// TIA Portal V18 export
DATA_BLOCK "06_Settings"   // DB8, F_DB
{ S7_Optimized_Access := 'TRUE'; DB_Accessible_From_OPC_UA := 'FALSE' }
// stored: DBAccessibleFromOPCUA false
   VAR
      Tristate : Bool;
      Reactivation_Delay : Time := T#10ms;
      Blink_Cyle_Time : Time := T#1S_260MS;
      ON_Time : Time := T#630MS;
      N_TRIG_RESET : Time;
   END_VAR
BEGIN
END_DATA_BLOCK
